// TIA Portal V17 export
// export: Created 2023-12-22T15:28:29.1657918Z, ExportSetting WithDefaults, DisplayName Totally Integrated Automation Portal, DisplayVersion V17, DisplayName TIA Portal Openness, DisplayVersion V17, DisplayName TIA Portal Version Control Interface, DisplayVersion V17, DisplayName STEP 7 Professional, DisplayVersion V17, DisplayName STEP 7 Safety, DisplayVersion V17, DisplayName WinCC Advanced, DisplayVersion V17
FUNCTION_BLOCK "ModBus_TCP"   // FB40, LAD
TITLE = Блок опроса ModBus TCP
{ S7_Optimized_Access := 'FALSE' }
VERSION : 0.1
// ВНИМАНИЕ!  Через один аппаратный порт контроллера можно проводить множество различных опросов по ModBus TCP. Для этого у каждого экземпляра должен быть указан уникальный CONNECT.ID.
// 
// Для каждого уникального CONNECT.ID / внешней ветки / точки подключения (IP, RemotePort) рекомендуется использовать отдельный экземпляр функционального блока. Например, при использовании tGW-735 имеющего 3 порта подключения с RemotePort = 502, 503 и 504 соответственно (но общий IP адрес) рекомендуется использовать три отдельных блока ModBus_TCP с уникальными CONNECT.ID.
// 
// Каждая точка чтения/записи = 1 экземпляр DEV_Config, количество элементов в массиве можно менять по необходимости, итоговое количество элементов массива указывается в теге Limit.
// 
// Для режима чтения необходимо указать:
// - MODE = 0
// - Source_DB = 40 (номер DB Modbus_TCP_DB)
// - SourceOFFSET = 0
// - Target_DB = xx (номер DB, куда необходимо положить прочитанные данные)
// - Target_OFFSET = xx (номер байта, начиная с которого кладутся прочитанные данные в выбранный DB)
// 
// Для режима опроса необходимо указать:
// - MODE = 1
// - Source_DB = xx (номер DB, откуда необходимо взять данные для передачи)
// - Source_OFFSET = xx (номер байта, начиная с которого берутся данные для передачи)
// - Target_DB = 40 (номер DB Modbus_TCP_DB)
// - Target_OFFSET = 0
// stored: AutoNumber false, IsIECCheckEnabled false, SetENOAutomatically false, UDAEnableTagReadback false
   VAR DB_SPECIFIC
      DATA : Array[0..100] of Word;   // Массив данных
      "Step" : Int;   // Шаг цикла опроса
      Device : Int := 1;   // Текущее устройство из списка DEV
      Limit { S7_SetPoint := 'True'} : Int := 10;   // Общее количество устройств
      COM_Control : Struct
         Enable { S7_SetPoint := 'True'} : Bool := true;   // Использовать коммуникацию
         Start : Bool;   // Начать опрос
         Reset : Bool;   // Сброс драйвера
         REQ_Done : Bool;   // Опрос завершён
         REQ_Busy : Bool;   // Опрос в процессе
         REQ_Error : Bool;   // Опрос - ошибка
         REQ_Status : Word;   // Опрос - код состояния
         Error_Code : Word;   // Опрос - код аварии
         Status : Int;   // 1 - успешно, 2 - нет ответа, 3 - ошибка параметров
      END_STRUCT;
      COM_REQ : Struct
         ADDR : UInt;   // Сетевой адрес устройства
         MODE : USInt;   // 0 - чтение, 1 - запись
         Register : UDInt;   // Начальный регистр опроса, см F1
         Length : UInt;   // Количество последовательных слов для опроса
      END_STRUCT;
      CONNECT { S7_SetPoint := 'True'} : TCON_IP_v4;
      DEV_Config : Array[1..10] of Struct
         Use { S7_SetPoint := 'True'} : Bool;   // 0 - не использовать, 1 - использовать
         MODE { S7_SetPoint := 'True'} : Bool;   // 0 - чтение, 1 - запись
         ADDR { S7_SetPoint := 'True'} : UInt;   // Сетевой адрес устройства
         Register { S7_SetPoint := 'True'} : UDInt;   // Начальный регистр опроса, см F1
         Length { S7_SetPoint := 'True'} : UInt;   // Количество последовательных слов для опроса
         Source_DB { S7_SetPoint := 'True'} : UInt;
         Source_OFFSET { S7_SetPoint := 'True'} : UInt;
         Target_DB { S7_SetPoint := 'True'} : UInt;
         Target_OFFSET { S7_SetPoint := 'True'} : UInt;
         Status : UInt;
      END_STRUCT;
   END_VAR
   VAR
      MB_CLIENT : MB_CLIENT;
      T_Busy : "Time_M";
   END_VAR
   // CONNECT.InterfaceId := 64;
   // CONNECT.ID := 16#0001;
   // CONNECT.ConnectionType := 16#0B;
   // CONNECT.ActiveEstablished := TRUE;
   // CONNECT.RemoteAddress.ADDR[1] := 16#C0;
   // CONNECT.RemoteAddress.ADDR[2] := 16#A8;
   // CONNECT.RemoteAddress.ADDR[3] := 16#00;
   // CONNECT.RemoteAddress.ADDR[4] := 16#0A;
   // CONNECT.RemotePort := 502;
   // CONNECT.LocalPort := 0;
   VAR_TEMP   // added for the SCL form of the ladder/FBD networks
      _w1 : Bool;
      _w2 : Bool;
      _w3 : Bool;
      _w4 : Bool;
      _w5 : Bool;
      _w6 : Bool;
      _w7 : Bool;
      _w8 : Bool;
      _w9 : Bool;
   END_VAR
BEGIN

REGION Network 1: Драйвер коммуникации
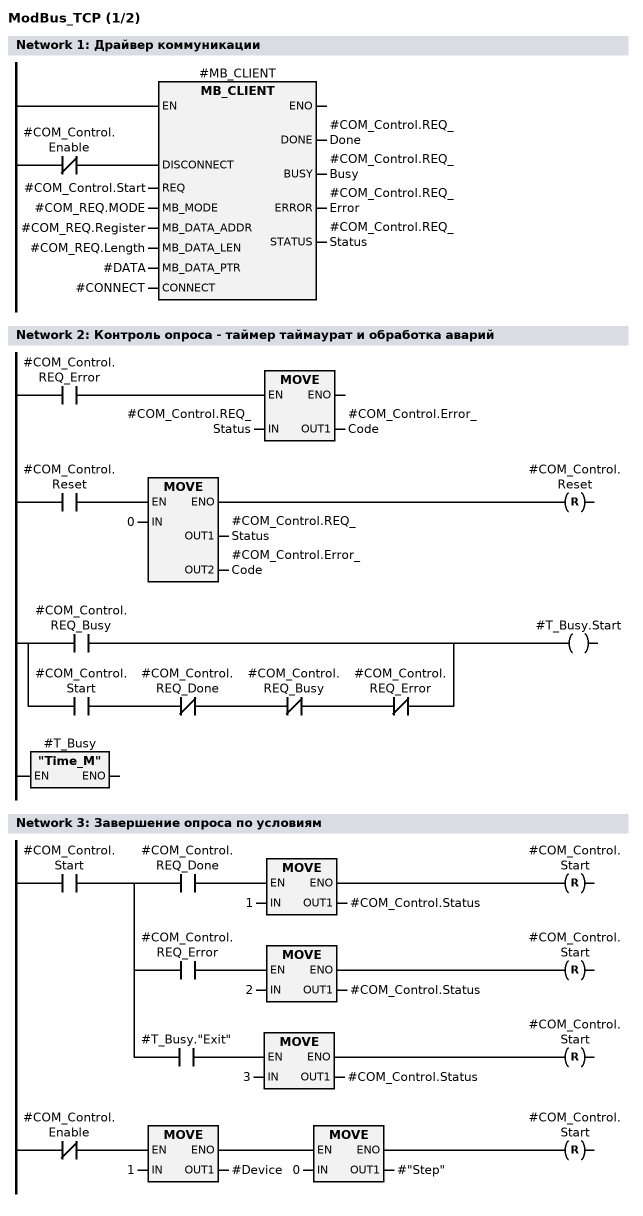
   RUNG wire#powerrail
      #MB_CLIENT.MB_CLIENT(DISCONNECT := wire#w1, REQ := #COM_Control.Start, MB_MODE := #COM_REQ.MODE, MB_DATA_ADDR := #COM_REQ.Register, MB_DATA_LEN := #COM_REQ.Length, MB_DATA_PTR := #DATA, CONNECT := #CONNECT, DONE => #COM_Control.REQ_Done, BUSY => #COM_Control.REQ_Busy, ERROR => #COM_Control.REQ_Error, STATUS => #COM_Control.REQ_Status)
   END_RUNG
   RUNG wire#powerrail
      I_Contact( #COM_Control.Enable )
   END_RUNG wire#w1
   // the same network as SCL:
   #MB_CLIENT(DISCONNECT := NOT #COM_Control.Enable,   // MB_CLIENT
              REQ := #COM_Control.Start,
              MB_MODE := #COM_REQ.MODE,
              MB_DATA_ADDR := #COM_REQ.Register,
              MB_DATA_LEN := #COM_REQ.Length,
              MB_DATA_PTR := #DATA,
              CONNECT := #CONNECT,
              DONE => #COM_Control.REQ_Done,
              BUSY => #COM_Control.REQ_Busy,
              ERROR => #COM_Control.REQ_Error,
              STATUS => #COM_Control.REQ_Status);
END_REGION

REGION Network 2: Контроль опроса - таймер таймаурат и обработка аварий
   RUNG wire#powerrail
      Contact( #COM_Control.REQ_Error )
      Move(in := #COM_Control.REQ_Status, out1 => #COM_Control.Error_Code)
   END_RUNG
   RUNG wire#powerrail
      Contact( #COM_Control.Reset )
      Move(in := 0, out1 => #COM_Control.REQ_Status, out2 => #COM_Control.Error_Code)
      R_Coil( #COM_Control.Reset )
   END_RUNG
   RUNG wire#powerrail
      Contact( #COM_Control.REQ_Busy )
      wire#w1
      Coil( #T_Busy.Start )
   END_RUNG
   RUNG wire#powerrail
      Contact( #COM_Control.Start )
      I_Contact( #COM_Control.REQ_Done )
      I_Contact( #COM_Control.REQ_Busy )
      I_Contact( #COM_Control.REQ_Error )
   END_RUNG wire#w1
   RUNG wire#powerrail
      #T_Busy()
   END_RUNG
   // the same network as SCL:
   IF #COM_Control.REQ_Error THEN #COM_Control.Error_Code := #COM_Control.REQ_Status; END_IF;
   IF #COM_Control.Reset THEN
       #COM_Control.REQ_Status := 0;
       #COM_Control.Error_Code := 0;
       #COM_Control.Reset := FALSE;
   END_IF;
   #T_Busy.Start := #COM_Control.REQ_Busy OR (#COM_Control.Start AND NOT #COM_Control.REQ_Done AND NOT #COM_Control.REQ_Busy AND NOT #COM_Control.REQ_Error);
   #T_Busy();   // "Time_M"
END_REGION

REGION Network 3: Завершение опроса по условиям
   RUNG wire#powerrail
      Contact( #COM_Control.Start )
      wire#w1
      Contact( #COM_Control.REQ_Done )
      Move(in := 1, out1 => #COM_Control.Status)
      R_Coil( #COM_Control.Start )
   END_RUNG
   RUNG wire#w1
      Contact( #COM_Control.REQ_Error )
      Move(in := 2, out1 => #COM_Control.Status)
      R_Coil( #COM_Control.Start )
   END_RUNG
   RUNG wire#w1
      Contact( #T_Busy."Exit" )
      Move(in := 3, out1 => #COM_Control.Status)
      R_Coil( #COM_Control.Start )
   END_RUNG
   RUNG wire#powerrail
      I_Contact( #COM_Control.Enable )
      Move(in := 1, out1 => #Device)
      Move(in := 0, out1 => #"Step")
      R_Coil( #COM_Control.Start )
   END_RUNG
   // the same network as SCL:
   IF #COM_Control.Start AND #COM_Control.REQ_Done THEN #COM_Control.Status := 1; END_IF;
   #_w1 := #COM_Control.Start;
   IF #COM_Control.Start AND #COM_Control.REQ_Done THEN #COM_Control.Start := FALSE; END_IF;
   IF #_w1 AND #COM_Control.REQ_Error THEN
       #COM_Control.Status := 2;
       #COM_Control.Start := FALSE;
   END_IF;
   IF #_w1 AND #T_Busy."Exit" THEN
       #COM_Control.Status := 3;
       #COM_Control.Start := FALSE;
   END_IF;
   IF NOT #COM_Control.Enable THEN
       #Device := 1;
       #"Step" := 0;
       #COM_Control.Start := FALSE;
   END_IF;
END_REGION

REGION Network 4: Цикл опроса активен
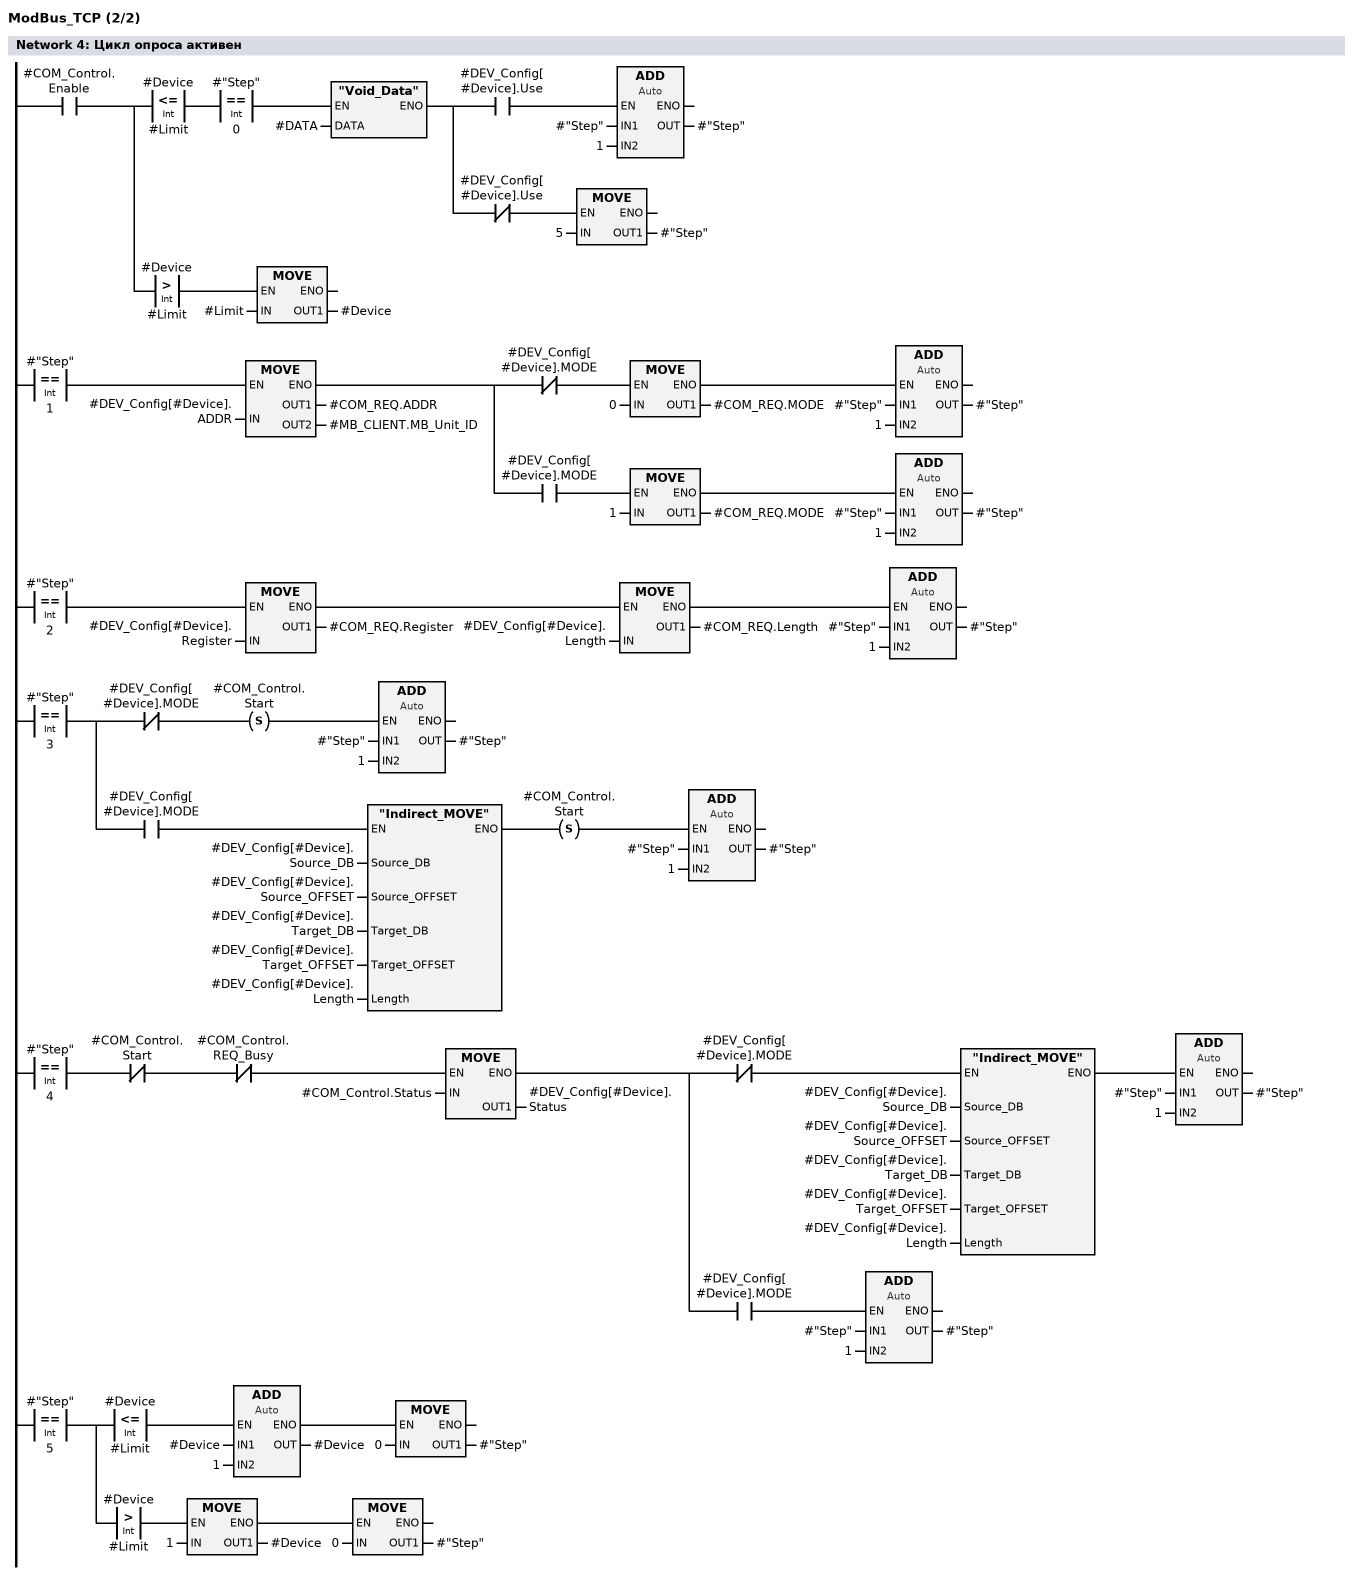
   RUNG wire#powerrail
      Contact( #COM_Control.Enable )
      wire#w1
      { S7_Templates := "SrcType := Int" } LE_Contact(in1 := #Device, in2 := #Limit)
      { S7_Templates := "SrcType := Int" } EQ_Contact(in1 := #"Step", in2 := 0)
      "Void_Data"(DATA := #DATA)
      wire#w2
      Contact( #DEV_Config[#Device].Use )
      Add(in1 := #"Step", in2 := 1, out => #"Step")
   END_RUNG
   RUNG wire#w2
      I_Contact( #DEV_Config[#Device].Use )
      Move(in := 5, out1 => #"Step")
   END_RUNG
   RUNG wire#w1
      { S7_Templates := "SrcType := Int" } GT_Contact(in1 := #Device, in2 := #Limit)
      Move(in := #Limit, out1 => #Device)
   END_RUNG
   RUNG wire#powerrail
      { S7_Templates := "SrcType := Int" } EQ_Contact(in1 := #"Step", in2 := 1)
      Move(in := #DEV_Config[#Device].ADDR, out1 => #COM_REQ.ADDR, out2 => #MB_CLIENT.MB_Unit_ID)
      wire#w3
      I_Contact( #DEV_Config[#Device].MODE )
      Move(in := 0, out1 => #COM_REQ.MODE)
      Add(in1 := #"Step", in2 := 1, out => #"Step")
   END_RUNG
   RUNG wire#w3
      Contact( #DEV_Config[#Device].MODE )
      Move(in := 1, out1 => #COM_REQ.MODE)
      Add(in1 := #"Step", in2 := 1, out => #"Step")
   END_RUNG
   RUNG wire#powerrail
      { S7_Templates := "SrcType := Int" } EQ_Contact(in1 := #"Step", in2 := 2)
      Move(in := #DEV_Config[#Device].Register, out1 => #COM_REQ.Register)
      Move(in := #DEV_Config[#Device].Length, out1 => #COM_REQ.Length)
      Add(in1 := #"Step", in2 := 1, out => #"Step")
   END_RUNG
   RUNG wire#powerrail
      { S7_Templates := "SrcType := Int" } EQ_Contact(in1 := #"Step", in2 := 3)
      wire#w4
      I_Contact( #DEV_Config[#Device].MODE )
      S_Coil( #COM_Control.Start )
      Add(in1 := #"Step", in2 := 1, out => #"Step")
   END_RUNG
   RUNG wire#w4
      Contact( #DEV_Config[#Device].MODE )
      "Indirect_MOVE"(Source_DB := #DEV_Config[#Device].Source_DB, Source_OFFSET := #DEV_Config[#Device].Source_OFFSET, Target_DB := #DEV_Config[#Device].Target_DB, Target_OFFSET := #DEV_Config[#Device].Target_OFFSET, Length := #DEV_Config[#Device].Length)
      S_Coil( #COM_Control.Start )
      Add(in1 := #"Step", in2 := 1, out => #"Step")
   END_RUNG
   RUNG wire#powerrail
      { S7_Templates := "SrcType := Int" } EQ_Contact(in1 := #"Step", in2 := 4)
      I_Contact( #COM_Control.Start )
      I_Contact( #COM_Control.REQ_Busy )
      Move(in := #COM_Control.Status, out1 => #DEV_Config[#Device].Status)
      wire#w5
      I_Contact( #DEV_Config[#Device].MODE )
      "Indirect_MOVE"(Source_DB := #DEV_Config[#Device].Source_DB, Source_OFFSET := #DEV_Config[#Device].Source_OFFSET, Target_DB := #DEV_Config[#Device].Target_DB, Target_OFFSET := #DEV_Config[#Device].Target_OFFSET, Length := #DEV_Config[#Device].Length)
      Add(in1 := #"Step", in2 := 1, out => #"Step")
   END_RUNG
   RUNG wire#w5
      Contact( #DEV_Config[#Device].MODE )
      Add(in1 := #"Step", in2 := 1, out => #"Step")
   END_RUNG
   RUNG wire#powerrail
      { S7_Templates := "SrcType := Int" } EQ_Contact(in1 := #"Step", in2 := 5)
      wire#w6
      { S7_Templates := "SrcType := Int" } LE_Contact(in1 := #Device, in2 := #Limit)
      Add(in1 := #Device, in2 := 1, out => #Device)
      Move(in := 0, out1 => #"Step")
   END_RUNG
   RUNG wire#w6
      { S7_Templates := "SrcType := Int" } GT_Contact(in1 := #Device, in2 := #Limit)
      Move(in := 1, out1 => #Device)
      Move(in := 0, out1 => #"Step")
   END_RUNG
   // the same network as SCL:
   "Void_Data"(EN := #COM_Control.Enable AND (#Device <= #Limit) AND (#"Step" = 0), DATA := #DATA, ENO => #_w1);
   IF #_w1 AND #DEV_Config[#Device].Use THEN #"Step" := #"Step" + 1; END_IF;
   IF #_w1 AND NOT #DEV_Config[#Device].Use THEN #"Step" := 5; END_IF;
   IF #COM_Control.Enable AND (#Device > #Limit) THEN #Device := #Limit; END_IF;
   #_w2 := #"Step" = 1;
   IF #_w2 THEN
       #COM_REQ.ADDR := #DEV_Config[#Device].ADDR;
       #MB_CLIENT.MB_Unit_ID := #DEV_Config[#Device].ADDR;
   END_IF;
   IF #_w2 AND NOT #DEV_Config[#Device].MODE THEN
       #COM_REQ.MODE := 0;
       #"Step" := #"Step" + 1;
   END_IF;
   IF #_w2 AND #DEV_Config[#Device].MODE THEN
       #COM_REQ.MODE := 1;
       #"Step" := #"Step" + 1;
   END_IF;
   IF #"Step" = 2 THEN
       #COM_REQ.Register := #DEV_Config[#Device].Register;
       #COM_REQ.Length := #DEV_Config[#Device].Length;
       #"Step" := #"Step" + 1;
   END_IF;
   #_w3 := #"Step" = 3;
   IF #_w3 AND NOT #DEV_Config[#Device].MODE THEN
       #COM_Control.Start := TRUE;
       #"Step" := #"Step" + 1;
   END_IF;
   "Indirect_MOVE"(EN := #_w3 AND #DEV_Config[#Device].MODE,
                   Source_DB := #DEV_Config[#Device].Source_DB,
                   Source_OFFSET := #DEV_Config[#Device].Source_OFFSET,
                   Target_DB := #DEV_Config[#Device].Target_DB,
                   Target_OFFSET := #DEV_Config[#Device].Target_OFFSET,
                   Length := #DEV_Config[#Device].Length,
                   ENO => #_w4);
   IF #_w4 THEN
       #COM_Control.Start := TRUE;
       #"Step" := #"Step" + 1;
   END_IF;
   #_w5 := (#"Step" = 4) AND NOT #COM_Control.Start AND NOT #COM_Control.REQ_Busy;
   IF #_w5 THEN #DEV_Config[#Device].Status := #COM_Control.Status; END_IF;
   "Indirect_MOVE"(EN := #_w5 AND NOT #DEV_Config[#Device].MODE,
                   Source_DB := #DEV_Config[#Device].Source_DB,
                   Source_OFFSET := #DEV_Config[#Device].Source_OFFSET,
                   Target_DB := #DEV_Config[#Device].Target_DB,
                   Target_OFFSET := #DEV_Config[#Device].Target_OFFSET,
                   Length := #DEV_Config[#Device].Length,
                   ENO => #_w6);
   IF #_w6 THEN #"Step" := #"Step" + 1; END_IF;
   IF #_w5 AND #DEV_Config[#Device].MODE THEN #"Step" := #"Step" + 1; END_IF;
   #_w7 := #"Step" = 5;
   #_w8 := #_w7 AND (#Device <= #Limit);
   IF #_w8 THEN
       #Device := #Device + 1;
       #"Step" := 0;
   END_IF;
   #_w9 := #_w7 AND (#Device > #Limit);
   IF #_w9 THEN
       #Device := 1;
       #"Step" := 0;
   END_IF;
END_REGION
END_FUNCTION_BLOCK
